// TIA Portal V19 export
TYPE "YourRecipeUDT"
   STRUCT
      "bool" : Bool;
      "int" : Int := 100;
      "dint" : DInt := 9876;
      "string" : String := 'a recipe';
   END_STRUCT;
END_TYPE
